(*
Casts I_Component to I_Signal
*)
FUNCTION ICompToISignal : Result
VAR_INPUT
	iSource	: I_Component;
END_VAR
VAR_OUTPUT
	iDest	: I_Signal;
END_VAR

IF iSource = 0 THEN
	ICompToISignal := Err.Itf0;
	RETURN;
END_IF

IF __QUERYINTERFACE(iSource, iDest) THEN
	ICompToISignal := Ok;
ELSE
	iDest := 0;
	ICompToISignal := Err.NoMatch;
END_IF

END_FUNCTION

(* stored: Version 1.1.0.1
   POU ICompToISignal: Id {5f959340-f887-4136-afe4-e25a563d68c5}, SpecialFunc None *)
